FUNCTION f_RobotNTCTengelytolTavol : BOOL

f_RobotNTCTengelytolTavol:=(GVL.stRobotStatusz.rX>-100) 
							OR (GVL.stRobotStatusz.rY>350)
							OR (GVL.stRobotStatusz.rZ>-111);

END_FUNCTION

(* stored: Version 1.1.0.1, ProductVersion 3.1.4024.11
   POU f_RobotNTCTengelytolTavol: Id {9ac71912-bbf0-4c31-b681-4766f05fa0ba}, SpecialFunc None *)
